TYPE ST_EL2809Ex EXTENDS ST_ReserveForGetSymbolNameByAddrress :
STRUCT
	Chl AT%Q* : ARRAY[1..16] OF BOOL;
END_STRUCT
END_TYPE

(* stored: Version 1.1.0.1, ProductVersion 3.1.4026.18
   DUT ST_EL2809Ex: Id {9e0bdd52-7fae-4317-9e8a-125993c10b1e} *)
